PROGRAM POU_3
VAR
END_VAR

END_PROGRAM

(* stored: Version 1.1.0.1, ProductVersion 3.1.4024.12
   POU POU_3: Id {3c04b035-fb99-4029-9ab8-cede714cb956}, SpecialFunc None *)
